// Mitsubishi GX Works2 project: 機電整合丙級第三題-ST   PLC: FX3U/FX3UC
// 機電整合丙級術科第三題ST語言版

// task Task_01 (event TRUE, interval 0, priority 31): POU_01

PROGRAM POU_01
VAR
  wProgramStep : INT;
  bM17 : BOOL;
  bM122 : BOOL;
  tmT122 : TIME;
  tdT122 : TON;
  wCountOf4 : INT;
  bM24 : BOOL;
  bM44 : BOOL;
  wC22 : INT;
END_VAR
(* 機電整合丙級術科第三題
   Author: Steven Luo
   Date: 2018/09/26
*)

IF M8002 OR NOT X17 THEN
	wProgramStep := 0;
	ZRST(TRUE, Y0, Y17);
	bM17 := FALSE;
	bM122 := FALSE;
END_IF;

IF NOT X17 THEN (* 按下急停 *)
	RST(TRUE, Y0);
	bM17 := TRUE;
END_IF;

IF X17 AND bM17 THEN (* 放開急停，等待復歸 *)
	wProgramStep := 122;
END_IF;

IF M8002 THEN
	wProgramStep := 21;
END_IF;

IF bM122 THEN
	IF M8013 THEN
		SET(TRUE, Y16); (* 黃燈閃爍 *)
	ELSE
		RST(TRUE, Y16);
	END_IF;
	tdT122(IN := TRUE, PT := T#3s); (* 計時三秒 *)
ELSE
	RST(TRUE, Y16);
END_IF;

CASE wProgramStep OF
	21:
		IF X1 AND NOT X5 AND X6 THEN
			SET(TRUE, Y17); (* 待機，綠燈亮、紅燈滅 *)
			RST(TRUE, Y15);
			wC22 := 0;
			wCountOf4 := 0;
			bM122 := FALSE;
			bM24 := FALSE;
			bM44 := FALSE;
		END_IF;
		IF X13 AND X17 AND X16 THEN (* 工作模式、按下啟動鈕 *)
			tdT122(IN := FALSE); (* tdT122的reset放在124似乎有問題，所以移到這裡 *)
			SET(TRUE, Y15); (* 紅燈亮、綠燈滅 *)
			RST(TRUE, Y17);
			wProgramStep := 22;
		END_IF;
	22:
		SET(TRUE, Y0); (* 推料缸伸出 *)
		INCP(X10, wC22); (* 啟動計數器 *)
		IF X0 THEN (* 推料缸前端點 *)
			IF wC22 = 2 THEN (* 凹槽在左 *)
				bM24 := TRUE;
				wProgramStep := 24;
			ELSE (* 凹槽在右 *)
				bM44 := TRUE;
				wProgramStep := 44;
			END_IF;
		END_IF;
	24:
		IF X3 OR X2 THEN
			SET(TRUE, Y4);
		END_IF;
		IF X4 THEN
			RST(TRUE, Y4);
			wProgramStep := 25;
		END_IF;
	25:
		SET(TRUE, Y7); (* 升降模組馬達旋轉 *)
		IF X7 THEN (* 升降模組下端點 *)
			RST(TRUE, Y7);
			IF X14 THEN (* 指定功能 *)
				IF X16 THEN
					wProgramStep := 26;
				END_IF;
			ELSE (* 單一循環 *)
				wProgramStep := 26;
			END_IF;
		END_IF;
	26:
		SET(TRUE, Y5); (* 真空吸盤吸 *)
		IF X5 THEN (* 壓力開關開 *)
			RST(TRUE, Y0); (* 推料缸退回 *)
			SET(TRUE, Y7); (* 升降模組馬達旋轉 *)
			IF X6 THEN (* 升降模組上端點 *)
				RST(TRUE, Y7);
				wProgramStep := 29;
			END_IF;
		END_IF;
	29:
		IF bM24 THEN (* 凹槽在左 *)
			SET(TRUE, Y3);
			IF X2 THEN
				RST(TRUE, Y3);
				wProgramStep := 210;
			END_IF;
		ELSIF bM44 THEN (* 凹槽在右 *)
			SET(TRUE, Y4);
			IF X2 THEN
				RST(TRUE, Y4);
				wProgramStep := 210;
			END_IF;
		END_IF;
	44:
		IF X4 OR X2 THEN
			SET(TRUE, Y3);
		END_IF;
		IF X3 THEN
			RST(TRUE, Y3);
			wProgramStep := 25;
		END_IF;
	122:
		IF NOT X13 AND X16 THEN (* 復歸模式、按下復歸開關 *)
			bM122 := TRUE;
			bM17 := FALSE;
			wProgramStep := 123;
		END_IF;
	123:
		IF NOT X6 THEN
			SET(TRUE, Y7); (* 升降模組馬達旋轉 *)
		END_IF;
		IF X6 THEN
			RST(TRUE, Y7);
			wProgramStep := 124;
		END_IF;
	124:
		IF X5 THEN
			SET(TRUE, Y6); (* 吸盤放 *)
		END_IF;
		IF NOT X5 THEN
			RST(TRUE, Y6);
		END_IF;
		IF tdT122.Q THEN
			wProgramStep := 21;
(*			tdT122(IN := FALSE);*)
		END_IF;
	210:
		SET(TRUE, Y7); (* 升降模組馬達旋轉 *)
		IF X7 THEN (* 升降模組下端點 *)
			RST(TRUE, Y7);
			IF NOT X14 OR (X14 AND X16) THEN
				RST(TRUE, Y5); (* 真空吸盤放 *)
				SET(TRUE, Y6);
				IF NOT X5 THEN
					RST(TRUE, Y6);
					wProgramStep := 211;
				END_IF;
			END_IF;
		END_IF;
	211:
		SET(TRUE, Y7); (* 升降模組馬達旋轉 *)
		IF X6 THEN (* 升降模組上端點 *)
			RST(TRUE, Y7);
			IF X15 AND (wCountOf4 < 3) THEN (* 連續循環 *)
				bM24 := FALSE;
				bM44 := FALSE;
				wC22 := 0;
				wCountOf4 := wCountOf4 + 1;
				wProgramStep := 22;
			ELSE (* 單一循環 *)
				wProgramStep := 21;
			END_IF;
		END_IF;
	ELSE
	;
END_CASE;
END_PROGRAM
